FUNCTION_BLOCK FB_InitialPressure
VAR_INPUT
	bEnable : BOOL;
	fCurrentPressure : LREAL;
END_VAR
VAR_OUTPUT
	fInitialPressure : LREAL;
END_VAR
VAR
END_VAR

IF bEnable THEN
	fInitialPressure := fInitialPressure;
ELSE 
	fInitialPressure := fCurrentPressure;
END_IF

END_FUNCTION_BLOCK

(* stored: Version 1.1.0.1, ProductVersion 3.1.4024.12
   POU FB_InitialPressure: Id {1da343e1-5d27-4580-a5e8-8e11a578ea02}, SpecialFunc None *)
